(* PLC project Untitled1, Beckhoff Automation GmbH TwinCAT PLC Control 3.5.13.20 *)
(* stored: creationDateTime 2022-07-20T15:23:00.1461411, modificationDateTime 2022-07-20T15:23:00.1461411 *)

{attribute 'qualified_only'}
{attribute 'strict'}
TYPE eFirmerVendorEvent3 : (eNoInfo := 0, eFanFault := 1, eStatisticsMemoryFault := 2, eRTCClockNotSet := 3, eRTCLowBatteryFault := 5, eRTCQuartzFault := 6);
END_TYPE
